Fanuc KAREL source: compact_preamble.KL

PROGRAM KB00110
%NOLOCKGROUP
%ENVIRONMENT IOSETUP
VAR
P1:INTEGER;P2:INTEGER;P3:INTEGER;P4:INTEGER
BEGIN
P1=1
P2=1
P3=1
P4=1
IO_MOD_TYPE(P1,P2,P3,P4)
END KB00110
